LIN {X 0,Y 67.21,Z 1184.367,A -85,B 0,C 180,E1 2334.022,E2 2334.022} C_VEL
LIN {X 0,Y 68.736,Z 1184.664,A -85,B 0,C 180,E1 2306.818,E2 2306.818} C_VEL
LIN {X 0,Y 54.608,Z 1187.245,A -85,B 0,C 180,E1 2287.19,E2 2287.19} C_VEL
LIN {X 0,Y 48.747,Z 1188.224,A -85,B 0,C 180,E1 2264.264,E2 2264.264} C_VEL
LIN {X 0,Y 48.12,Z 1188.423,A -85,B 0,C 180,E1 2248.824,E2 2248.824} C_VEL
LIN {X 0,Y 49.322,Z 1188.169,A -85,B 0,C 180,E1 2231.088,E2 2231.088} C_VEL
LIN {X 0,Y 57.401,Z 1186.721,A -85,B 0,C 180,E1 2207.224,E2 2207.224} C_VEL
LIN {X 0,Y 71.86,Z 1184.107,A -85,B 0,C 180,E1 2190.401,E2 2190.401} C_VEL
LIN {X 0,Y 92.62,Z 1179.572,A -85,B 0,C 180,E1 2178.22,E2 2178.22} C_VEL
LIN {X 0,Y 114.958,Z 1173.749,A -85,B 0,C 180,E1 2170.663,E2 2170.663} C_VEL
LIN {X 0,Y 139.567,Z 1165.803,A -85,B 0,C 180,E1 2165.299,E2 2165.299} C_VEL
LIN {X 0,Y 164.03,Z 1156.49,A -85,B 0,C 180,E1 2161.583,E2 2161.583} C_VEL
LIN {X 0,Y 170.979,Z 1153.609,A -85,B 0,C 180,E1 2160.705,E2 2160.705} C_VEL
LIN {X 0,Y 148.099,Z 1163.373,A -85,B 0,C 180,E1 2157.603,E2 2157.603} C_VEL
LIN {X 0,Y 122.927,Z 1172.511,A -85,B 0,C 180,E1 2152.856,E2 2152.856} C_VEL
LIN {X 0,Y 101.62,Z 1179.067,A -85,B 0,C 180,E1 2146.899,E2 2146.899} C_VEL
LIN {X 0,Y 80.214,Z 1184.523,A -85,B 0,C 180,E1 2137.259,E2 2137.259} C_VEL
LIN {X 0,Y 62.322,Z 1188.439,A -85,B 0,C 180,E1 2122.117,E2 2122.117} C_VEL
LIN {X 0,Y 57.198,Z 1189.386,A -85,B 0,C 180,E1 2116.596,E2 2116.596} C_VEL
LIN {X 0,Y 46.528,Z 1190.545,A -85,B 0,C 180,E1 2104.718,E2 2104.718} C_VEL
LIN {X 0,Y 41.468,Z 1190.958,A -85,B 0,C 180,E1 2093.308,E2 2093.308} C_VEL
LIN {X 0,Y 40.802,Z 1191.027,A -85,B 0,C 180,E1 2089.52,E2 2089.52} C_VEL
LIN {X 0,Y 40.103,Z 1191.317,A -85,B 0,C 180,E1 2071.411,E2 2071.411} C_VEL
LIN {X 0,Y 40.346,Z 1191.113,A -85,B 0,C 180,E1 2055.633,E2 2055.633} C_VEL
LIN {X 0,Y 46.549,Z 1190.01,A -85,B 0,C 180,E1 2028.23,E2 2028.23} C_VEL
LIN {X 0,Y 62.701,Z 1187.158,A -85,B 0,C 180,E1 2006.52,E2 2006.52} C_VEL
LIN {X 0,Y 73.13,Z 1185.094,A -85,B 0,C 180,E1 1999.157,E2 1999.157} C_VEL
LIN {X 0,Y 58.666,Z 1185.603,A -85,B 0,C 180,E1 1971.176,E2 1971.176} C_VEL
LIN {X 0,Y 59.91,Z 1185.764,A -85,B 0,C 180,E1 1948.842,E2 1948.842} C_VEL
LIN {X 0,Y 45.471,Z 1187.852,A -85,B 0,C 180,E1 1926.44,E2 1926.44} C_VEL
LIN {X 0,Y 40.559,Z 1188.539,A -85,B 0,C 180,E1 1902.837,E2 1902.837} C_VEL
LIN {X 0,Y 40.131,Z 1188.666,A -85,B 0,C 180,E1 1887.161,E2 1887.161} C_VEL
LIN {X 0,Y 41.99,Z 1188.406,A -85,B 0,C 180,E1 1866.139,E2 1866.139} C_VEL
LIN {X 0,Y 52.29,Z 1186.901,A -85,B 0,C 180,E1 1840.125,E2 1840.125} C_VEL
LIN {X 0,Y 70.48,Z 1184.022,A -85,B 0,C 180,E1 1822.786,E2 1822.786} C_VEL
LIN {X 0,Y 92.342,Z 1179.426,A -85,B 0,C 180,E1 1812.507,E2 1812.507} C_VEL
LIN {X 0,Y 116.59,Z 1173.195,A -85,B 0,C 180,E1 1805.896,E2 1805.896} C_VEL
LIN {X 0,Y 140.675,Z 1165.641,A -85,B 0,C 180,E1 1801.629,E2 1801.629} C_VEL
LIN {X 0,Y 146.845,Z 1163.458,A -85,B 0,C 180,E1 1800.729,E2 1800.729} C_VEL
LIN {X 0,Y 121.731,Z 1172.315,A -85,B 0,C 180,E1 1796.704,E2 1796.704} C_VEL
LIN {X 0,Y 98.171,Z 1179.287,A -85,B 0,C 180,E1 1791.048,E2 1791.048} C_VEL
LIN {X 0,Y 75.642,Z 1184.573,A -85,B 0,C 180,E1 1782.096,E2 1782.096} C_VEL
LIN {X 0,Y 56.11,Z 1188.416,A -85,B 0,C 180,E1 1767.002,E2 1767.002} C_VEL
LIN {X 0,Y 43.563,Z 1190.468,A -85,B 0,C 180,E1 1743.407,E2 1743.407} C_VEL
LIN {X 0,Y 40.802,Z 1191.027,A -85,B 0,C 180,E1 1729.52,E2 1729.52} C_VEL
LIN {X 0,Y 39.335,Z 1191.153,A -85,B 0,C 180,E1 1721.093,E2 1721.093} C_VEL
LIN {X 0,Y 36.611,Z 1191.206,A -85,B 0,C 180,E1 1709.117,E2 1709.117} C_VEL
LIN {X 0,Y 34.705,Z 1190.569,A -85,B 0,C 180,E1 1678.384,E2 1678.384} C_VEL
LIN {X 0,Y 35.66,Z 1190.381,A -85,B 0,C 180,E1 1673.956,E2 1673.956} C_VEL
LIN {X 0,Y 48.948,Z 1188.539,A -85,B 0,C 180,E1 1648.524,E2 1648.524} C_VEL
LIN {X 0,Y 61.835,Z 1186.46,A -85,B 0,C 180,E1 1637.742,E2 1637.742} C_VEL
LIN {X 0,Y 50.065,Z 1186.753,A -85,B 0,C 180,E1 1602.568,E2 1602.568} C_VEL
LIN {X 0,Y 51.16,Z 1186.708,A -85,B 0,C 180,E1 1591.609,E2 1591.609} C_VEL
LIN {X 0,Y 37.19,Z 1188.341,A -85,B 0,C 180,E1 1568.221,E2 1568.221} C_VEL
LIN {X 0,Y 32.372,Z 1188.855,A -85,B 0,C 180,E1 1540.702,E2 1540.702} C_VEL
LIN {X 0,Y 32.214,Z 1188.892,A -85,B 0,C 180,E1 1522.89,E2 1522.89} C_VEL
LIN {X 0,Y 35.848,Z 1188.509,A -85,B 0,C 180,E1 1496.117,E2 1496.117} C_VEL
LIN {X 0,Y 48.137,Z 1187.082,A -85,B 0,C 180,E1 1471.639,E2 1471.639} C_VEL
LIN {X 0,Y 68.586,Z 1184.156,A -85,B 0,C 180,E1 1455.846,E2 1455.846} C_VEL
LIN {X 0,Y 91.692,Z 1179.58,A -85,B 0,C 180,E1 1447.164,E2 1447.164} C_VEL
LIN {X 0,Y 118.075,Z 1172.956,A -85,B 0,C 180,E1 1441.456,E2 1441.456} C_VEL
LIN {X 0,Y 121.983,Z 1171.844,A -85,B 0,C 180,E1 1440.751,E2 1440.751} C_VEL
LIN {X 0,Y 96.79,Z 1179.087,A -85,B 0,C 180,E1 1435.853,E2 1435.853} C_VEL
LIN {X 0,Y 72.586,Z 1184.466,A -85,B 0,C 180,E1 1427.92,E2 1427.92} C_VEL
LIN {X 0,Y 50.445,Z 1188.342,A -85,B 0,C 180,E1 1413.087,E2 1413.087} C_VEL
LIN {X 0,Y 36.53,Z 1190.255,A -85,B 0,C 180,E1 1388.991,E2 1388.991} C_VEL
LIN {X 0,Y 32.13,Z 1190.966,A -85,B 0,C 180,E1 1358.929,E2 1358.929} C_VEL
LIN {X 0,Y 32.085,Z 1191.022,A -85,B 0,C 180,E1 1345.757,E2 1345.757} C_VEL
LIN {X 0,Y 34.889,Z 1190.505,A -85,B 0,C 180,E1 1316.984,E2 1316.984} C_VEL
LIN {X 0,Y 35.66,Z 1190.381,A -85,B 0,C 180,E1 1313.956,E2 1313.956} C_VEL
LIN {X 0,Y 37.107,Z 1190.057,A -85,B 0,C 180,E1 1306.077,E2 1306.077} C_VEL
LIN {X 0,Y 40.822,Z 1188.928,A -85,B 0,C 180,E1 1285.425,E2 1285.425} C_VEL
LIN {X 0,Y 43.83,Z 1188.471,A -85,B 0,C 180,E1 1280.913,E2 1280.913} C_VEL
LIN {X 0,Y 50.398,Z 1187.642,A -85,B 0,C 180,E1 1275.438,E2 1275.438} C_VEL
LIN {X 0,Y 42.418,Z 1187.57,A -85,B 0,C 180,E1 1235.381,E2 1235.381} C_VEL
LIN {X 0,Y 27.079,Z 1188.981,A -85,B 0,C 180,E1 1203.664,E2 1203.664} C_VEL
LIN {X 0,Y 24.134,Z 1189.204,A -85,B 0,C 180,E1 1172.404,E2 1172.404} C_VEL
LIN {X 0,Y 25.631,Z 1189.043,A -85,B 0,C 180,E1 1144.619,E2 1144.619} C_VEL
LIN {X 0,Y 38.026,Z 1188.094,A -85,B 0,C 180,E1 1109.843,E2 1109.843} C_VEL
LIN {X 0,Y 59.345,Z 1185.495,A -85,B 0,C 180,E1 1092.311,E2 1092.311} C_VEL
LIN {X 0,Y 84.871,Z 1181.176,A -85,B 0,C 180,E1 1083.377,E2 1083.377} C_VEL
LIN {X 0,Y 96.497,Z 1178.778,A -85,B 0,C 180,E1 1080.838,E2 1080.838} C_VEL
LIN {X 0,Y 71.305,Z 1184.174,A -85,B 0,C 180,E1 1074.515,E2 1074.515} C_VEL
LIN {X 0,Y 47.27,Z 1188.055,A -85,B 0,C 180,E1 1062.099,E2 1062.099} C_VEL
LIN {X 0,Y 30.592,Z 1189.985,A -85,B 0,C 180,E1 1038.706,E2 1038.706} C_VEL
LIN {X 0,Y 24.192,Z 1190.701,A -85,B 0,C 180,E1 1001.896,E2 1001.896} C_VEL
LIN {X 0,Y 24.087,Z 1190.765,A -85,B 0,C 180,E1 985.064,E2 985.064} C_VEL
LIN {X 0,Y 28.572,Z 1190.213,A -85,B 0,C 180,E1 947.298,E2 947.298} C_VEL
LIN {X 0,Y 43.83,Z 1188.471,A -85,B 0,C 180,E1 920.913,E2 920.913} C_VEL
LIN {X 0,Y 44.648,Z 1188.278,A -85,B 0,C 180,E1 918.367,E2 918.367} C_VEL
LIN {X 0,Y 43.99,Z 1188.151,A -85,B 0,C 180,E1 914.47,E2 914.47} C_VEL
LIN {X 0,Y 41.508,Z 1188.141,A -85,B 0,C 180,E1 908.749,E2 908.749} C_VEL
LIN {X 0,Y 34.621,Z 1188.402,A -85,B 0,C 180,E1 891.065,E2 891.065} C_VEL
LIN {X 0,Y 34.295,Z 1188.406,A -85,B 0,C 180,E1 887.911,E2 887.911} C_VEL
LIN {X 0,Y 34.063,Z 1188.397,A -85,B 0,C 180,E1 881.266,E2 881.266} C_VEL
LIN {X 0,Y 18.227,Z 1189.322,A -85,B 0,C 180,E1 843.314,E2 843.314} C_VEL
LIN {X 0,Y 16.141,Z 1189.473,A -85,B 0,C 180,E1 806.492,E2 806.492} C_VEL
LIN {X 0,Y 20.791,Z 1189.255,A -85,B 0,C 180,E1 763.881,E2 763.881} C_VEL
LIN {X 0,Y 39.163,Z 1187.913,A -85,B 0,C 180,E1 734.102,E2 734.102} C_VEL
LIN {X 0,Y 62.066,Z 1185.286,A -85,B 0,C 180,E1 723.025,E2 723.025} C_VEL
LIN {X 0,Y 69.347,Z 1184.186,A -85,B 0,C 180,E1 720.869,E2 720.869} C_VEL
LIN {X 0,Y 43.514,Z 1187.983,A -85,B 0,C 180,E1 711.033,E2 711.033} C_VEL
LIN {X 0,Y 24.396,Z 1189.846,A -85,B 0,C 180,E1 689.336,E2 689.336} C_VEL
LIN {X 0,Y 16.15,Z 1190.484,A -85,B 0,C 180,E1 640.66,E2 640.66} C_VEL
LIN {X 0,Y 16.098,Z 1190.502,A -85,B 0,C 180,E1 622.82,E2 622.82} C_VEL
LIN {X 0,Y 23.68,Z 1189.903,A -85,B 0,C 180,E1 572.328,E2 572.328} C_VEL
LIN {X 0,Y 39.162,Z 1188.459,A -85,B 0,C 180,E1 551.786,E2 551.786} C_VEL
LIN {X 0,Y 34.295,Z 1188.406,A -85,B 0,C 180,E1 527.911,E2 527.911} C_VEL
LIN {X 0,Y 33.159,Z 1188.484,A -85,B 0,C 180,E1 524.183,E2 524.183} C_VEL
LIN {X 0,Y 30.393,Z 1188.647,A -85,B 0,C 180,E1 520.801,E2 520.801} C_VEL
LIN {X 0,Y 25.489,Z 1188.952,A -85,B 0,C 180,E1 517.854,E2 517.854} C_VEL
LIN {X 0,Y 14.924,Z 1189.537,A -85,B 0,C 180,E1 511.407,E2 511.407} C_VEL
LIN {X 0,Y 11.98,Z 1189.594,A -85,B 0,C 180,E1 502.97,E2 502.97} C_VEL
LIN {X 0,Y 8.168,Z 1189.735,A -85,B 0,C 180,E1 443.056,E2 443.056} C_VEL
LIN {X 0,Y 16.254,Z 1189.523,A -85,B 0,C 180,E1 382.785,E2 382.785} C_VEL
LIN {X 0,Y 38.998,Z 1188.108,A -85,B 0,C 180,E1 361.581,E2 361.581} C_VEL
LIN {X 0,Y 40.251,Z 1187.997,A -85,B 0,C 180,E1 361.079,E2 361.079} C_VEL
LIN {X 0,Y 16.862,Z 1189.889,A -85,B 0,C 180,E1 341.443,E2 341.443} C_VEL
LIN {X 0,Y 8.106,Z 1190.279,A -85,B 0,C 180,E1 269.913,E2 269.913} C_VEL
LIN {X 0,Y 16.883,Z 1189.88,A -85,B 0,C 180,E1 198.507,E2 198.507} C_VEL
LIN {X 0,Y 28.237,Z 1189.082,A -85,B 0,C 180,E1 184.57,E2 184.57} C_VEL
LIN {X 0,Y 26.336,Z 1188.994,A -85,B 0,C 180,E1 170.961,E2 170.961} C_VEL
LIN {X 0,Y 11.98,Z 1189.594,A -85,B 0,C 180,E1 142.97,E2 142.97} C_VEL
LIN {X 0,Y 9.189,Z 1189.681,A -85,B 0,C 180,E1 131.618,E2 131.618} C_VEL
LIN {X 0,Y 4.172,Z 1189.866,A -85,B 0,C 180,E1 100.898,E2 100.898} C_VEL
LIN {X 0,Y 2.125,Z 1189.946,A -85,B 0,C 180,E1 39.059,E2 39.059} C_VEL
LIN {X 0,Y 1.474,Z 1189.99,A -85,B 0,C 180,E1 2.4,E2 2.4} C_VEL
LIN {X 0,Y 1.394,Z 1189.987,A -85,B 0,C 180,E1 177.836,E2 177.836} C_VEL
LIN {X 0,Y 1.474,Z 1189.99,A -85,B 0,C 180,E1 2.4,E2 2.4} C_VEL
LIN {X 0,Y 3.501,Z 1191.99,A -85,B 0,C 180,E1 -1.765,E2 -1.765} C_VEL
LIN {X 0,Y 3.501,Z 1215,A -85,B 0,C 180,E1 -1.765,E2 -1.765} C_VEL
LIN {X 0,Y 3.501,Z 1215,A -85,B 0,C 180,E1 -1.765,E2 -1.765}

QRS_NEXT_CUT()

QRS_NEXT()
QRS_HOME()

END
